# EPICS substitutions: products/ITER/products/org.csstudio.iter.css.product/demo/m-TEST-BOY/src/main/epics/SharedTemplateApp/Db/ramp.substitutions
file ramp.db {
    pattern { IOC, COUNT, SCAN }
        { "A", "0", ".2 second" }
        { "A", "1", ".2 second" }
        { "A", "2", ".2 second" }
        { "A", "3", ".2 second" }
        { "A", "4", ".2 second" }
        { "A", "5", ".2 second" }
        { "A", "6", ".2 second" }
        { "A", "7", ".2 second" }
        { "A", "8", ".2 second" }
        { "A", "9", ".2 second" }
        { "A", "10", ".2 second" }
        { "A", "11", ".2 second" }
        { "A", "12", ".2 second" }
        { "A", "13", ".2 second" }
        { "A", "14", ".2 second" }
        { "A", "15", ".2 second" }
        { "A", "16", ".2 second" }
        { "A", "17", ".2 second" }
        { "A", "18", ".2 second" }
        { "A", "19", ".2 second" }
        { "A", "20", ".2 second" }
        { "A", "21", ".2 second" }
        { "A", "22", ".2 second" }
        { "A", "23", ".2 second" }
        { "A", "24", ".2 second" }
        { "A", "25", ".2 second" }
        { "A", "26", ".2 second" }
        { "A", "27", ".2 second" }
        { "A", "28", ".2 second" }
        { "A", "29", ".2 second" }
        { "A", "30", ".2 second" }
        { "A", "31", ".2 second" }
        { "A", "32", ".2 second" }
        { "A", "33", ".2 second" }
        { "A", "34", ".2 second" }
        { "A", "35", ".2 second" }
        { "A", "36", ".2 second" }
        { "A", "37", ".2 second" }
        { "A", "38", ".2 second" }
        { "A", "39", ".2 second" }
        { "A", "40", ".2 second" }
        { "A", "41", ".2 second" }
        { "A", "42", ".2 second" }
        { "A", "43", ".2 second" }
        { "A", "44", ".2 second" }
        { "A", "45", ".2 second" }
        { "A", "46", ".2 second" }
        { "A", "47", ".2 second" }
        { "A", "48", ".2 second" }
        { "A", "49", ".2 second" }
        { "A", "50", ".2 second" }
        { "A", "51", ".2 second" }
        { "A", "52", ".2 second" }
        { "A", "53", ".2 second" }
        { "A", "54", ".2 second" }
        { "A", "55", ".2 second" }
        { "A", "56", ".2 second" }
        { "A", "57", ".2 second" }
        { "A", "58", ".2 second" }
        { "A", "59", ".2 second" }
        { "A", "60", ".2 second" }
        { "A", "61", ".2 second" }
        { "A", "62", ".2 second" }
        { "A", "63", ".2 second" }
        { "A", "64", ".2 second" }
        { "A", "65", ".2 second" }
        { "A", "66", ".2 second" }
        { "A", "67", ".2 second" }
        { "A", "68", ".2 second" }
        { "A", "69", ".2 second" }
        { "A", "70", ".2 second" }
        { "A", "71", ".2 second" }
        { "A", "72", ".2 second" }
        { "A", "73", ".2 second" }
        { "A", "74", ".2 second" }
        { "A", "75", ".2 second" }
        { "A", "76", ".2 second" }
        { "A", "77", ".2 second" }
        { "A", "78", ".2 second" }
        { "A", "79", ".2 second" }
        { "A", "80", ".2 second" }
        { "A", "81", ".2 second" }
        { "A", "82", ".2 second" }
        { "A", "83", ".2 second" }
        { "A", "84", ".2 second" }
        { "A", "85", ".2 second" }
        { "A", "86", ".2 second" }
        { "A", "87", ".2 second" }
        { "A", "88", ".2 second" }
        { "A", "89", ".2 second" }
        { "A", "90", ".2 second" }
        { "A", "91", ".2 second" }
        { "A", "92", ".2 second" }
        { "A", "93", ".2 second" }
        { "A", "94", ".2 second" }
        { "A", "95", ".2 second" }
        { "A", "96", ".2 second" }
        { "A", "97", ".2 second" }
        { "A", "98", ".2 second" }
        { "A", "99", ".2 second" }
        { "A", "100", ".2 second" }
        { "A", "101", ".2 second" }
        { "A", "102", ".2 second" }
        { "A", "103", ".2 second" }
        { "A", "104", ".2 second" }
        { "A", "105", ".2 second" }
        { "A", "106", ".2 second" }
        { "A", "107", ".2 second" }
        { "A", "108", ".2 second" }
        { "A", "109", ".2 second" }
        { "A", "110", ".2 second" }
        { "A", "111", ".2 second" }
        { "A", "112", ".2 second" }
        { "A", "113", ".2 second" }
        { "A", "114", ".2 second" }
        { "A", "115", ".2 second" }
        { "A", "116", ".2 second" }
        { "A", "117", ".2 second" }
        { "A", "118", ".2 second" }
        { "A", "119", ".2 second" }
        { "A", "120", ".2 second" }
        { "A", "121", ".2 second" }
        { "A", "122", ".2 second" }
        { "A", "123", ".2 second" }
        { "A", "124", ".2 second" }
        { "A", "125", ".2 second" }
        { "A", "126", ".2 second" }
        { "A", "127", ".2 second" }
        { "A", "128", ".2 second" }
        { "A", "129", ".2 second" }
        { "A", "130", ".2 second" }
        { "A", "131", ".2 second" }
        { "A", "132", ".2 second" }
        { "A", "133", ".2 second" }
        { "A", "134", ".2 second" }
        { "A", "135", ".2 second" }
        { "A", "136", ".2 second" }
        { "A", "137", ".2 second" }
        { "A", "138", ".2 second" }
        { "A", "139", ".2 second" }
        { "A", "140", ".2 second" }
        { "A", "141", ".2 second" }
        { "A", "142", ".2 second" }
        { "A", "143", ".2 second" }
        { "A", "144", ".2 second" }
        { "A", "145", ".2 second" }
        { "A", "146", ".2 second" }
        { "A", "147", ".2 second" }
        { "A", "148", ".2 second" }
        { "A", "149", ".2 second" }
        { "A", "150", ".2 second" }
        { "A", "151", ".2 second" }
        { "A", "152", ".2 second" }
        { "A", "153", ".2 second" }
        { "A", "154", ".2 second" }
        { "A", "155", ".2 second" }
        { "A", "156", ".2 second" }
        { "A", "157", ".2 second" }
        { "A", "158", ".2 second" }
        { "A", "159", ".2 second" }
        { "A", "160", ".2 second" }
        { "A", "161", ".2 second" }
        { "A", "162", ".2 second" }
        { "A", "163", ".2 second" }
        { "A", "164", ".2 second" }
        { "A", "165", ".2 second" }
        { "A", "166", ".2 second" }
        { "A", "167", ".2 second" }
        { "A", "168", ".2 second" }
        { "A", "169", ".2 second" }
        { "A", "170", ".2 second" }
        { "A", "171", ".2 second" }
        { "A", "172", ".2 second" }
        { "A", "173", ".2 second" }
        { "A", "174", ".2 second" }
        { "A", "175", ".2 second" }
        { "A", "176", ".2 second" }
        { "A", "177", ".2 second" }
        { "A", "178", ".2 second" }
        { "A", "179", ".2 second" }
        { "A", "180", ".2 second" }
        { "A", "181", ".2 second" }
        { "A", "182", ".2 second" }
        { "A", "183", ".2 second" }
        { "A", "184", ".2 second" }
        { "A", "185", ".2 second" }
        { "A", "186", ".2 second" }
        { "A", "187", ".2 second" }
        { "A", "188", ".2 second" }
        { "A", "189", ".2 second" }
        { "A", "190", ".2 second" }
        { "A", "191", ".2 second" }
        { "A", "192", ".2 second" }
        { "A", "193", ".2 second" }
        { "A", "194", ".2 second" }
        { "A", "195", ".2 second" }
        { "A", "196", ".2 second" }
        { "A", "197", ".2 second" }
        { "A", "198", ".2 second" }
        { "A", "199", ".2 second" }
}
